FUNCTION_BLOCK AQ_TO_AB (* Converts an AQ (Quarter Byte) adapter to an AB (BYTE) adapter *)
  (* Standard: 61499-2; Description: Copyright (c) 2026 Meisterschulen am Ostbahnhof SPDX-License-Identifier: EPL-2.0 *)
  (* Version 1.0, 2026-05-16, Franz Höpfinger, Meisterschulen am Ostbahnhof, Initial Version *)
  PACKAGE adapter::conversion::unidirectional;
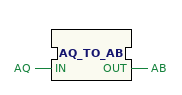
  SOCKETS
    IN : adapter::types::unidirectional::AQ; (* AQ Input *)
  END_SOCKETS
  PLUGS
    OUT : adapter::types::unidirectional::AB; (* BYTE Output *)
  END_PLUGS
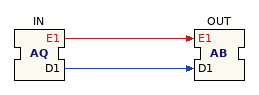
  EVENT_CONNECTIONS
    IN.E1 TO OUT.E1;
  END_CONNECTIONS
  DATA_CONNECTIONS
    IN.D1 TO OUT.D1;
  END_CONNECTIONS
END_FUNCTION_BLOCK
